{attribute 'linkalways'} 
{attribute 'no_explicit_call' := 'This FB is a CLASS and must be accessed using methods or properties'}
{attribute 'enable_dynamic_creation'}
FUNCTION_BLOCK FINAL AND_WORD EXTENDS Node
VAR
	in1 : _WORD(0);
	in2 : _WORD(0);
	out : _WORD(0);
END_VAR

METHOD PUBLIC Clone : I_Node
VAR
	pNode : POINTER TO AND_WORD;
END_VAR
pNode := __NEW(AND_WORD);
Clone := pNode^;
END_METHOD

METHOD FB_init : BOOL
VAR_INPUT
	bInitRetains : BOOL; // if TRUE, the retain variables are initialized (warm start / cold start)
	bInCopyCode : BOOL;  // if TRUE, the instance afterwards gets moved into the copy code (online change)
END_VAR
AddInput('in1',THIS^.in1);
AddInput('in2',THIS^.in2);
AddOutput('out', THIS^.out);
END_METHOD

METHOD PROTECTED OnExecute
VAR
END_VAR
out.Value := in1.Value AND in2.Value;
END_METHOD

END_FUNCTION_BLOCK

(* stored: Version 1.1.0.1, ProductVersion 3.1.4024.15
   POU AND_WORD: Id {5acbfbdf-96b7-4370-97c0-024dde4d1c81}, SpecialFunc None
   Folder Constructor: Id {51cf803a-bd6f-4b31-a0fb-38ba655696a8}
   Method Clone: Id {5fe4b01c-4004-44d5-909a-4512b176c679}
   Method FB_init: Id {148afbfd-20a9-49ac-9b3a-fce19f02f8ef}
   Method OnExecute: Id {3e40d7fe-3aed-455c-93cb-f1d2a7722436} *)
